TYPE ST_ValveOutputs :
STRUCT
	bEnable AT %I* : BOOL;
	nValveOut AT %Q* : INT;
END_STRUCT
END_TYPE

(* stored: Version 1.1.0.1, ProductVersion 3.1.4024.12
   DUT ST_ValveOutputs: Id {2a8c6fb8-d112-4222-97fe-ebaee0ecbde4} *)
